// TwinCAT 3 PLC project PLC
// ProgramVersion: 3.1.4024.0
// libraries:
//   Tc2_Standard, * (Beckhoff Automation GmbH)
//   Tc2_System, * (Beckhoff Automation GmbH)
//   Tc3_Module, * (Beckhoff Automation GmbH)
// project tree:
//   DUTs/ S_TestStruct.TcDUT
//   GVLs/ GK.TcGVL, GM.TcGVL
//   / PlcTask.TcTTO
//   POUs/ MAIN.TcPOU
// real-time tasks:
//   TASK PlcTask: cycle T#10ms, priority 20, ADS port 350

CONFIGURATION PLC
    RESOURCE PLC ON TwinCAT3
        TASK PlcTask(INTERVAL := T#10ms, PRIORITY := 20);
        PROGRAM MAIN WITH PlcTask : MAIN;
    END_RESOURCE
END_CONFIGURATION

// ---- DUTs/S_TestStruct.TcDUT
TYPE S_TestStruct :
STRUCT
	fReal : REAL;
	nInt : INT;
	bBit : BOOL;
END_STRUCT
END_TYPE

// ---- GVLs/GK.TcGVL
{attribute 'qualified_only'}
VAR_GLOBAL
	
	// A string to test reading.
	sReadTest : STRING := 'The quick brown fox jumps over the lazy dog.';
	
END_VAR

// ---- GVLs/GM.TcGVL
{attribute 'qualified_only'}
VAR_GLOBAL
	
	// Simulated bit value.
	bBit : BOOL;
	// Simulated integer value.
	nInteger : INT;
	// Simulated real value.
	fReal : REAL;
	
	// Target string variable to test writing strings.
	sTarget : T_MaxString;
	
	// A string that will echo the value of sTarget to test reading back strings.
	sEcho : T_MaxString;
	
	jit : _Implicit_Jitter_Distribution;
	
	stTestStruct : S_TestStruct;
	
	aTestArray : ARRAY [ 0 .. 9 ] OF REAL;
	
END_VAR

// ---- POUs/MAIN.TcPOU
PROGRAM MAIN
VAR
	// Alternates between TRUE and FALSE on a 1 second tick.
	bBlink : BOOL;
	// Timer for the blink variable.
	tonBlink : TON;
	
	nArrayIndex : INT;
END_VAR


tonBlink(IN:=TRUE, PT:=T#1S);
IF tonBlink.Q THEN
	
	bBlink := NOT bBlink;
	
	GM.bBit := NOT GM.bBit;
	GM.nInteger := GM.nInteger + 1;	
	GM.fReal := LREAL_TO_REAL(SIN(GM.nInteger) * 10);
	GM.sEcho := GM.sTarget;
	
	tonBlink(IN:=FALSE);
	
	
	GM.stTestStruct.bBit := NOT GM.bBit;
	GM.stTestStruct.nInt := 16000 - GM.nInteger;
	GM.stTestStruct.fReal := COS(GM.fReal) * 100;
	
	nArrayIndex := GM.nInteger MOD 10;
	GM.aTestArray[nArrayIndex] := TAN(GM.fReal);
	
END_IF

END_PROGRAM
